// TIA Portal V20 export
FUNCTION "FC1_SelfHold" : Void   // FC36, LAD
TITLE = FC1_SelfHold
{ S7_Optimized_Access := 'TRUE' }
// Set/Reset 코일을 사용하지 않는 자기유지(Self-Holding) 회로
// stored: SetENOAutomatically false
   VAR_INPUT
      Input1 : Bool;
      Input2 : Bool;
   END_VAR
   VAR_OUTPUT
      Output1 : Bool;
   END_VAR
BEGIN

REGION Network 1: 자기유지 회로
   // (Input1 OR Output1) AND NOT Input2 -> Output1
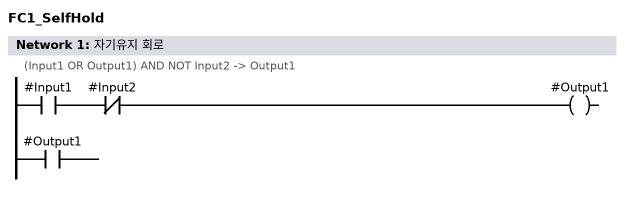
   #Output1 := #Input1 AND NOT #Input2;
END_REGION
END_FUNCTION
